// TIA Portal V18 export
FUNCTION "calc_speeds_from_mechanics_2SyncedDrivesTUBEZ" : Void   // FC25, FBD
{ S7_Optimized_Access := 'TRUE' }
VERSION : 0.1
// stored: AutoNumber true, IsIECCheckEnabled false, SetENOAutomatically false, UDAEnableTagReadback false
   VAR_INPUT
      mm_per_outputshaft_rev : Real;
      reduction_ration : Real;
      max_revs_at_10V : Real;
      counts_per_encoder_rev : Real;
      encoder_placed_on_motor : Bool;
   END_VAR
   VAR_OUTPUT
      Vabsmax_mm_per_s : Real;
      counts_per_mm : Real;
      ER_params : Bool;
   END_VAR
   VAR_IN_OUT
      para : "typeMotPara";
   END_VAR
   VAR_TEMP
      t_acceleration_s : Real;
      maxV_mm_per_min : Real;
      "a" : Real;
      v_abs_max : Real;
      t_mx : Real;
      dist_fast : Real;
      v_min_viable : Real;
      dist_stop : Real;
      dist_auto_done : Real;
      K_min : Real;
      K_min_dist : Real;
      dist_absMax : Real;
      t_fst : Real;
      v_fast : Real;
   END_VAR
BEGIN

REGION Network 2 (SCL)

   #maxV_mm_per_min := #max_revs_at_10V / #reduction_ration * #mm_per_outputshaft_rev;

   #Vabsmax_mm_per_s := #maxV_mm_per_min / 60;
END_REGION

REGION Network 3 (SCL)
   IF #encoder_placed_on_motor THEN
       #counts_per_mm :=  #counts_per_encoder_rev * #reduction_ration / #mm_per_outputshaft_rev  ;
   ELSE
       #counts_per_mm := #counts_per_encoder_rev /  #mm_per_outputshaft_rev;

   END_IF;
END_REGION

REGION Network 4 (SCL)
   #v_abs_max := #Vabsmax_mm_per_s;
   #t_acceleration_s := #para.t_acc_50Hz_USER;
   #v_fast := #para.v_absoluteMax_LOGIC;

   #K_min := 1.0/50.0;
   #v_min_viable := #v_abs_max * #K_min;

   #t_mx := #t_acceleration_s;
   #ER_params := #t_acceleration_s = 0 OR #v_abs_max = 0 OR #t_mx =0 ;
   IF NOT #ER_params THEN
       #t_fst := #t_acceleration_s * #v_fast / #v_abs_max;
       #a := #v_abs_max / #t_mx;
       #dist_absMax := #a * #t_mx * #t_mx / 2 + #v_min_viable * #t_mx;
       #dist_fast := #a * #t_fst * #t_fst / 2 + #v_min_viable * #t_fst;
   ELSE
       #a := 0;
       #dist_fast := #dist_absMax := 999;
       #t_fst := 0;
   END_IF;
   #K_min_dist := 1.0/ 50.0;//#K_min * 0.8;
   #dist_stop := #dist_absMax * #K_min_dist;
   #dist_auto_done := #dist_stop * 4.0;//1.4;//.0;// 1.2;
END_REGION

REGION Network 5 (SCL)
   #para.dist_absMax_LOGIC := #dist_fast;
   #para.dist_stop_USER := #dist_stop;
   #para.dist_auto_done_LOGIC := #dist_auto_done;
   #para.v_absoluteMax_LOGIC := #v_abs_max;
   #para.v_crawl_USER := #v_min_viable;
END_REGION
END_FUNCTION
